TYPE UNIT_Blikkenvullijn_SIM :
STRUCT
	Starting_SC 	: BOOL;
	Execute_SC 		: BOOL;
	Resetting_SC 	: BOOL;
	Holding_SC 		: BOOL;
	Unholding_SC 	: BOOL;
	Suspending_SC	: BOOL;
	Unsuspending_SC	: BOOL;
	Aborting_SC		: BOOL;
	Clearing_SC		: BOOL;
	Stopping_SC		: BOOL;
END_STRUCT
END_TYPE

(* stored: Version 1.1.0.1, ProductVersion 3.1.4024.12
   DUT UNIT_Blikkenvullijn_SIM: Id {b367c448-e25a-4eed-97da-83609ecbd1fb} *)
